// TIA Portal V16 export
// export: Created 2024-09-05T15:58:42.6122143Z, ExportSetting WithDefaults, DisplayName Totally Integrated Automation Portal, DisplayVersion V16 Update 6, DisplayName TIA Portal Version Control Interface, DisplayVersion V16 Update 2, DisplayName TIA Portal Openness, DisplayVersion V16 Update 6, DisplayName STEP 7 Professional, DisplayVersion V16 Update 6, DisplayName STEP 7 Safety, DisplayVersion V16, DisplayName WinCC Advanced, DisplayVersion V16 Update 6
VAR_GLOBAL   // PLC tag table "R1 sensors"
   iR1tubePresentFront AT %I22.0 : Bool;
   iR1tubePresentRear AT %I22.1 : Bool;
END_VAR
